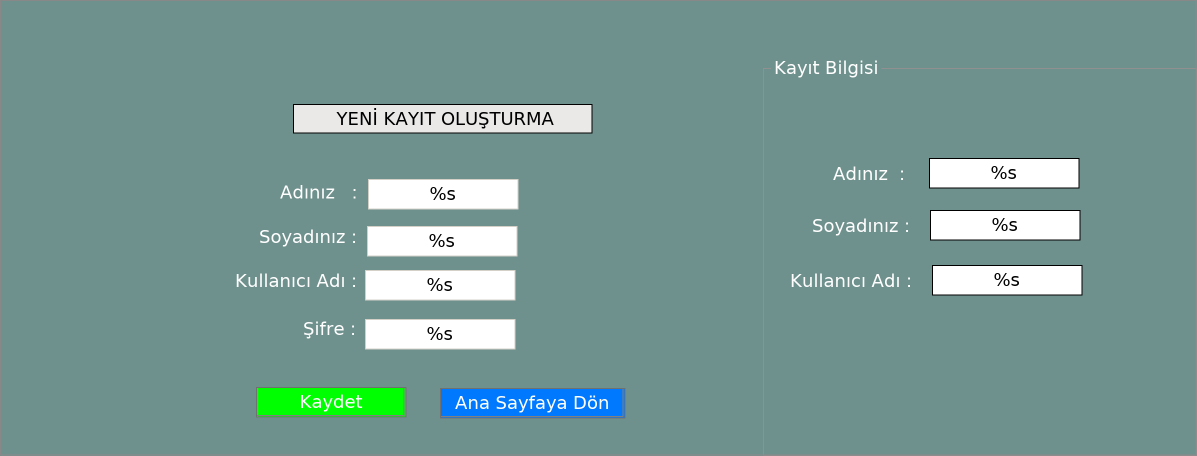
VISUALIZATION uyelik_sayfa  // 1197x456
    Rectangle (293,104 299x29)
    Label (244,176 150x33), "Adınız :"
    Label (233,222 150x30), "Soyadınız :"
    Label (216,265 160x32), "Kullanıcı Adı :"
    Label (255,315 149x28), "Şifre :"
    Label (311,104 269x30), "YENİ KAYIT OLUŞTURMA"
    Textfield (368,179 150x30), "%s", text variable: MAIN.ad
        OnMouseClick: write the text variable via Edit
    Textfield (367,226 150x30), "%s", text variable: MAIN.soyad
        OnMouseClick: write the text variable via Edit
    Textfield (365,319 150x30), "%s", text variable: MAIN.yenisifre
        OnMouseClick: write the text variable via Edit
    Textfield (365,270 150x30), "%s", text variable: MAIN.yenikul
        OnMouseClick: write the text variable via Edit
    Button (256,387 150x30), "Kaydet"
        tap MAIN.kaydet
        OnMouseClick: OpenDialog Dialog=VisuDialogs.MessageBox, Parameters={eType: MAIN.msgtype, sMessageTxt: MAIN.msgtxt, sTitle: MAIN.msgtitle}, OpenModal=True, OpenCentered=True
    Button (440,388 185x30), "Ana Sayfaya Dön"
        OnMouseClick: change screen: Ana_Sayfa
    GroupBox (763,60 434x396), "Kayıt Bilgisi"
        Rectangle (166,98 150x30), "%s", text variable: MAIN.ad
        Label (38,99 136x30), "Adınız :"
        Label (23,151 150x30), "Soyadınız :"
        Rectangle (167,150 150x30), "%s", text variable: MAIN.soyad
        Label (13,206 150x30), "Kullanıcı Adı :"
        Rectangle (169,205 150x30), "%s", text variable: MAIN.yenikul
END_VISUALIZATION

(* stored: Version 1.1.0.1, ProductVersion 3.1.4024.12
   Visu uyelik_sayfa: Id {92c37705-9ee6-492e-80c5-5cfa0db86768} *)
